# EPICS autosave request: iocBoot/gmca_23b_ioc2/dbSave/XZ_P11_.req
%
% BURT Request File
%
% $(P)XZ:P10:  X-Y positioner #11
%

file assy.req ASSY=$(P)XZ:P11
file mtr1.req MTR1=$(P)XZ:mx11
file mtr1.req MTR1=$(P)XZ:my11
file drv1.req DRV1=$(P)XZ:X11
file drv1.req DRV1=$(P)XZ:Y11
